// Mitsubishi GX Works2 project: MiniFactory   PLC: FX2N/FX2NC

PROGRAM MAIN
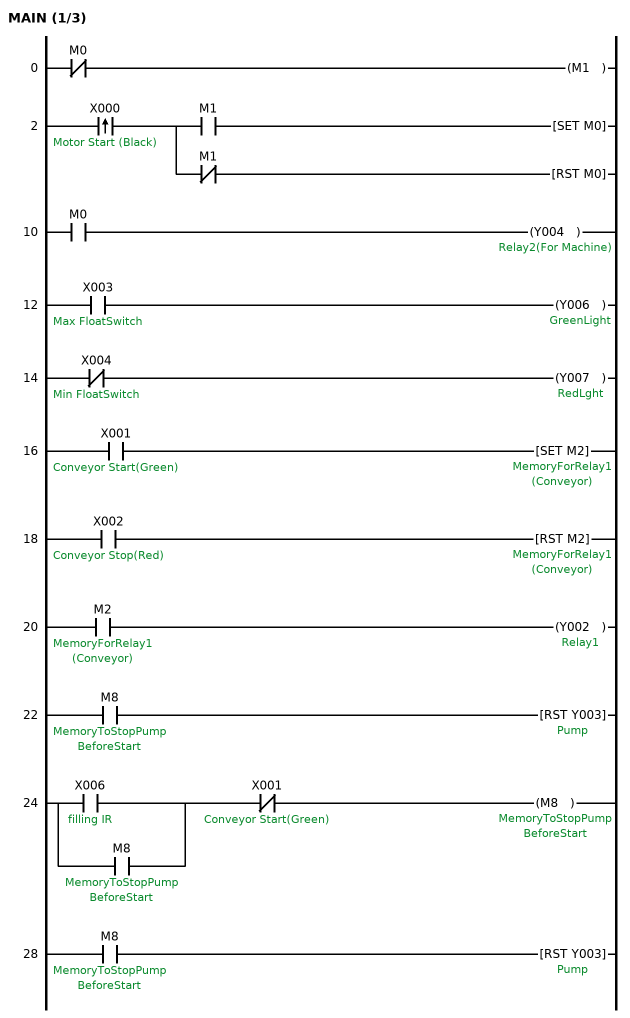
0     LDI     M0
      OUT     M1
2     LDP     X000  ; Motor Start (Black)
      MPS
      AND     M1
      SET     M0
      MPP
      ANI     M1
      RST     M0
10    LD      M0
      OUT     Y004  ; Relay2(For Machine)
12    LD      X003  ; Max FloatSwitch
      OUT     Y006  ; GreenLight
14    LDI     X004  ; Min FloatSwitch
      OUT     Y007  ; RedLght
16    LD      X001  ; Conveyor Start(Green)
      SET     M2  ; MemoryForRelay1 (Conveyor)
18    LD      X002  ; Conveyor Stop(Red)
      RST     M2  ; MemoryForRelay1 (Conveyor)
20    LD      M2  ; MemoryForRelay1 (Conveyor)
      OUT     Y002  ; Relay1
22    LD      M8  ; MemoryToStopPumpBeforeStart
      RST     Y003  ; Pump
24    LD      X006  ; filling IR
      OR      M8  ; MemoryToStopPumpBeforeStart
      ANI     X001  ; Conveyor Start(Green)
      OUT     M8  ; MemoryToStopPumpBeforeStart
28    LD      M8  ; MemoryToStopPumpBeforeStart
      RST     Y003  ; Pump
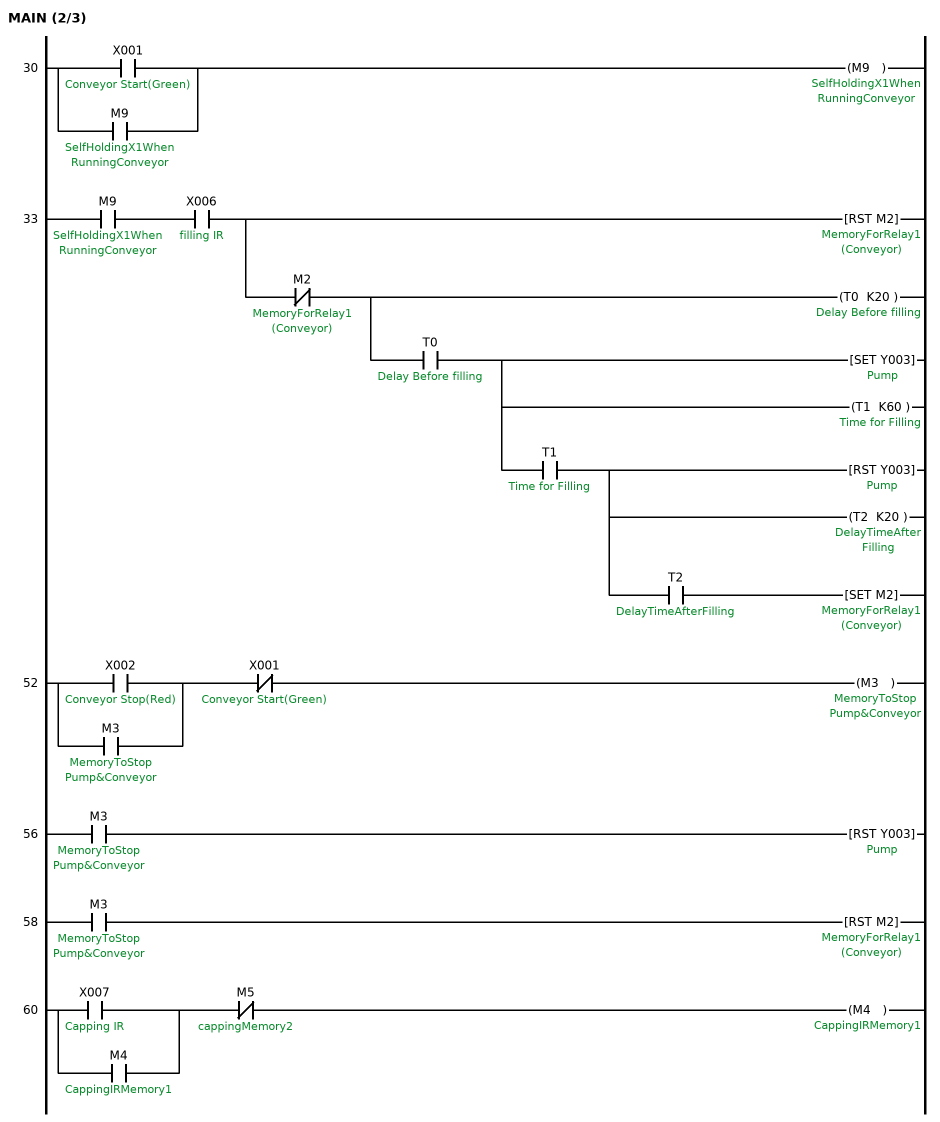
30    LD      X001  ; Conveyor Start(Green)
      OR      M9  ; SelfHoldingX1WhenRunningConveyor
      OUT     M9  ; SelfHoldingX1WhenRunningConveyor
33    LD      M9  ; SelfHoldingX1WhenRunningConveyor
      AND     X006  ; filling IR
      RST     M2  ; MemoryForRelay1 (Conveyor)
      ANI     M2  ; MemoryForRelay1 (Conveyor)
      OUT     T0 K20  ; Delay Before filling
      AND     T0  ; Delay Before filling
      SET     Y003  ; Pump
      OUT     T1 K60  ; Time for Filling
      AND     T1  ; Time for Filling
      RST     Y003  ; Pump
      OUT     T2 K20  ; DelayTimeAfterFilling
      AND     T2  ; DelayTimeAfterFilling
      SET     M2  ; MemoryForRelay1 (Conveyor)
52    LD      X002  ; Conveyor Stop(Red)
      OR      M3  ; MemoryToStopPump&Conveyor
      ANI     X001  ; Conveyor Start(Green)
      OUT     M3  ; MemoryToStopPump&Conveyor
56    LD      M3  ; MemoryToStopPump&Conveyor
      RST     Y003  ; Pump
58    LD      M3  ; MemoryToStopPump&Conveyor
      RST     M2  ; MemoryForRelay1 (Conveyor)
60    LD      X007  ; Capping IR
      OR      M4  ; CappingIRMemory1
      ANI     M5  ; cappingMemory2
      OUT     M4  ; CappingIRMemory1
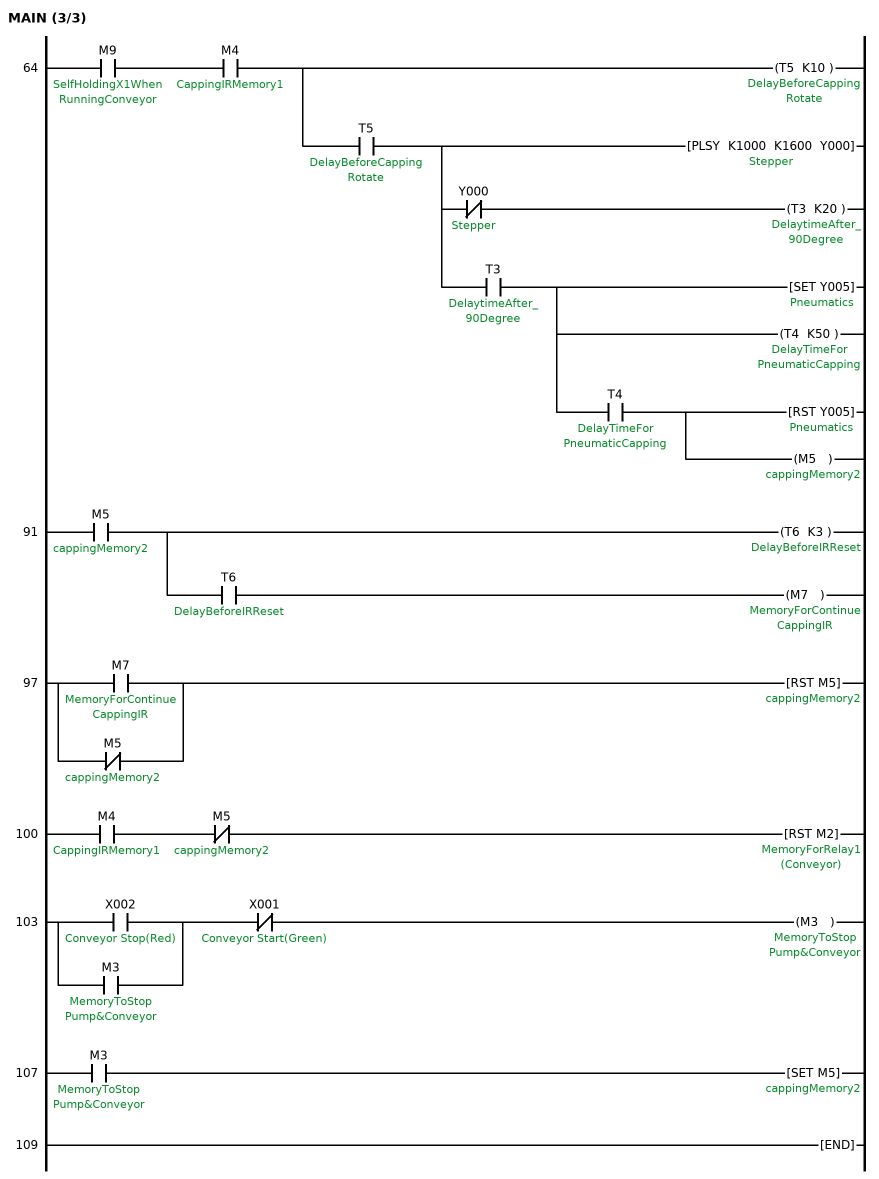
64    LD      M9  ; SelfHoldingX1WhenRunningConveyor
      AND     M4  ; CappingIRMemory1
      OUT     T5 K10  ; DelayBeforeCappingRotate
      AND     T5  ; DelayBeforeCappingRotate
      PLSY    K1000 K1600 Y000  ; Stepper
      MPS
      ANI     Y000  ; Stepper
      OUT     T3 K20  ; DelaytimeAfter_90Degree
      MPP
      AND     T3  ; DelaytimeAfter_90Degree
      SET     Y005  ; Pneumatics
      OUT     T4 K50  ; DelayTimeForPneumaticCapping
      AND     T4  ; DelayTimeForPneumaticCapping
      RST     Y005  ; Pneumatics
      OUT     M5  ; cappingMemory2
91    LD      M5  ; cappingMemory2
      OUT     T6 K3  ; DelayBeforeIRReset
      AND     T6  ; DelayBeforeIRReset
      OUT     M7  ; MemoryForContinueCappingIR
97    LD      M7  ; MemoryForContinueCappingIR
      ORI     M5  ; cappingMemory2
      RST     M5  ; cappingMemory2
100   LD      M4  ; CappingIRMemory1
      ANI     M5  ; cappingMemory2
      RST     M2  ; MemoryForRelay1 (Conveyor)
103   LD      X002  ; Conveyor Stop(Red)
      OR      M3  ; MemoryToStopPump&Conveyor
      ANI     X001  ; Conveyor Start(Green)
      OUT     M3  ; MemoryToStopPump&Conveyor
107   LD      M3  ; MemoryToStopPump&Conveyor
      SET     M5  ; cappingMemory2
109   END
END_PROGRAM

// device comments not shown above
X005  ; filling IR
Y001  ; Red Light
M6  ; MemoryToResetIR
